/// This enumeration contains all steps that are used by the various sequences of a unit.
/// Sequences use a subrange (***Begin to ***End) of this enumeration.
{attribute 'qualified_only'}
{attribute 'to_string'}
TYPE AssemblyStep :
(
  Undefined := 0
  
  ,BootBegin
  ,BootEnd 

  ,StopBegin
  ,StopEnd

  ,AutomaticBegin
  ,AutomaticEnd
  
  ,GoHomeBegin
  ,GoHomeGoToHomePos
  ,GoHomeEnd 
  
  ,FaultReactionBegin
  ,FaultReactionEnd
);
END_TYPE

(* stored: Version 1.1.0.1
   DUT AssemblyStep: Id {f5e137a4-3c70-4dba-810c-35b6df03ecce} *)
